// TIA Portal V20 export
FUNCTION_BLOCK "LER_SimHmiRotaryAxis"   // FB13, LAD
// stored: Access Published, MemoryReserve 100, SetENOAutomatically false
   VAR_INPUT
      axisActualPos { ExternalAccessible := 'False'; ExternalVisible := 'False'; ExternalWritable := 'False'} : LReal;
      referenceDesignator { ExternalAccessible := 'False'; ExternalVisible := 'False'; ExternalWritable := 'False'} : WString;
   END_VAR
   VAR_OUTPUT
      simHmiAxis { ExternalAccessible := 'False'; ExternalVisible := 'False'; ExternalWritable := 'False'} : "LER_typeSimRotaryAxis";
   END_VAR
   VAR
      statPrePosition { ExternalAccessible := 'False'; ExternalVisible := 'False'; ExternalWritable := 'False'} : LReal;
   END_VAR
BEGIN

REGION Network 2
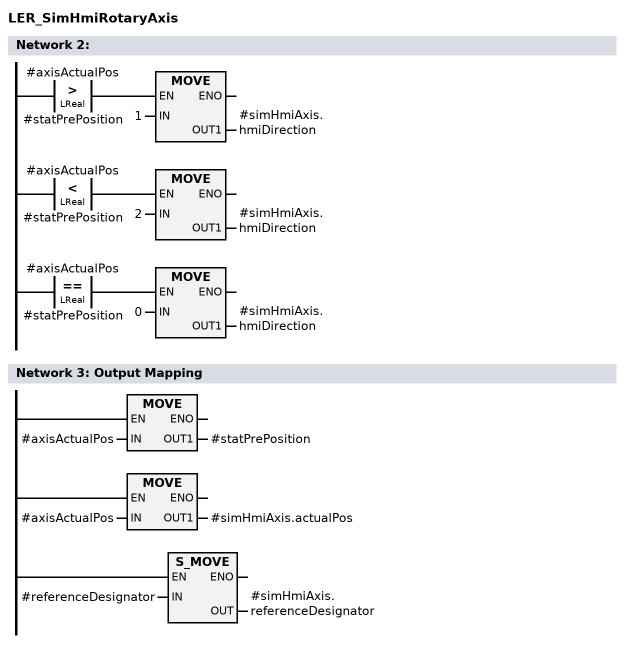
   RUNG wire#powerrail
      { S7_Templates := "SrcType := LReal" } GT_Contact(in1 := #axisActualPos, in2 := #statPrePosition)
      Move(in := 1, out1 => #simHmiAxis.hmiDirection)
   END_RUNG
   RUNG wire#powerrail
      { S7_Templates := "SrcType := LReal" } LT_Contact(in1 := #axisActualPos, in2 := #statPrePosition)
      Move(in := 2, out1 => #simHmiAxis.hmiDirection)
   END_RUNG
   RUNG wire#powerrail
      { S7_Templates := "SrcType := LReal" } EQ_Contact(in1 := #axisActualPos, in2 := #statPrePosition)
      Move(in := 0, out1 => #simHmiAxis.hmiDirection)
   END_RUNG
   // the same network as SCL:
   IF #axisActualPos > #statPrePosition THEN #simHmiAxis.hmiDirection := 1; END_IF;
   IF #axisActualPos < #statPrePosition THEN #simHmiAxis.hmiDirection := 2; END_IF;
   IF #axisActualPos = #statPrePosition THEN #simHmiAxis.hmiDirection := 0; END_IF;
END_REGION

REGION Network 3: Output Mapping
   RUNG wire#powerrail
      Move(in := #axisActualPos, out1 => #statPrePosition)
   END_RUNG
   RUNG wire#powerrail
      Move(in := #axisActualPos, out1 => #simHmiAxis.actualPos)
   END_RUNG
   RUNG wire#powerrail
      S_Move(in := #referenceDesignator, out => #simHmiAxis.referenceDesignator)
   END_RUNG
   // the same network as SCL:
   #statPrePosition := #axisActualPos;
   #simHmiAxis.actualPos := #axisActualPos;
   #simHmiAxis.referenceDesignator := #referenceDesignator;
END_REGION
END_FUNCTION_BLOCK
